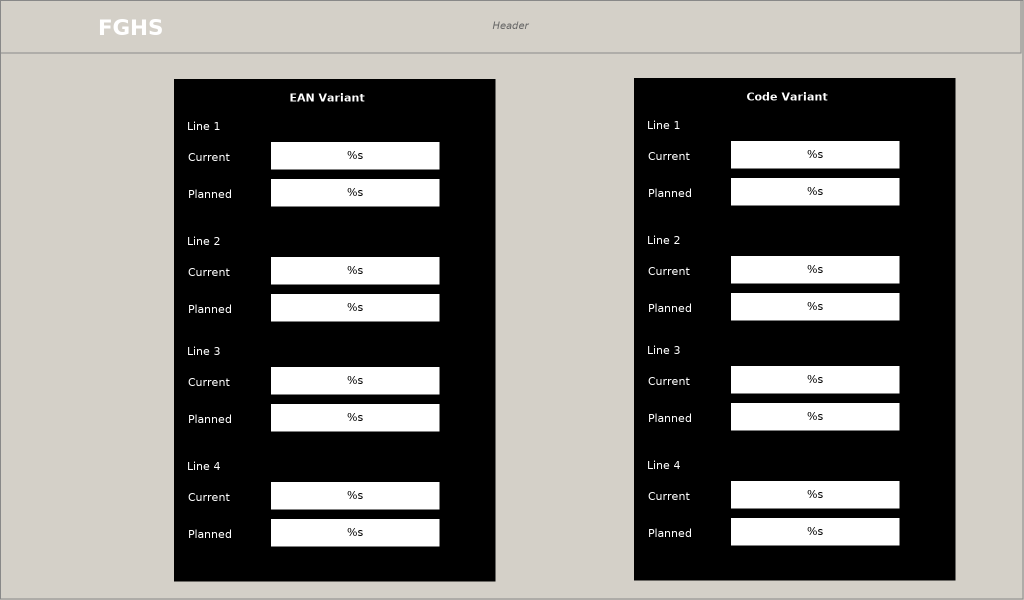
VISUALIZATION FGHS_1  // 1024x600
    Frame (0,-2 1021x55)
        shows Header()
    RoundedRectangle (174,79 321x502)
    Label (214,78 227x40), "EAN Variant"
    Label (185,140 78x35), "Current"
    RoundedRectangle (270,141 170x29), "%s", text variable: Status_GVL.arCurrent_EAN[1]
        OnMouseClick: write Status_GVL.RecipeLine[1].EANVariant via Default
    Label (185,177 78x35), "Planned"
    RoundedRectangle (270,178 170x29), "%s", text variable: Status_GVL.arPlanned_EAN[1]
    Label (95,15 250x25), "FGHS"
    Label (184,109 78x35), "Line 1"
    Label (185,255 78x35), "Current"
    RoundedRectangle (270,256 170x29), "%s", text variable: Status_GVL.arCurrent_EAN[2]
        OnMouseClick: write Status_GVL.RecipeLine[2].EANVariant via Default
    Label (185,292 78x35), "Planned"
    RoundedRectangle (270,293 170x29), "%s", text variable: Status_GVL.arPlanned_EAN[2]
    Label (184,224 78x35), "Line 2"
    Label (185,365 78x35), "Current"
    RoundedRectangle (270,366 170x29), "%s", text variable: Status_GVL.arCurrent_EAN[3]
        OnMouseClick: write Status_GVL.RecipeLine[3].EANVariant via Default
    Label (185,402 78x35), "Planned"
    RoundedRectangle (270,403 170x29), "%s", text variable: Status_GVL.arPlanned_EAN[3]
    Label (184,334 78x35), "Line 3"
    Label (185,480 78x35), "Current"
    RoundedRectangle (270,481 170x29), "%s", text variable: Status_GVL.arCurrent_EAN[4]
        OnMouseClick: write Status_GVL.RecipeLine[4].EANVariant via Default
    Label (185,517 78x35), "Planned"
    RoundedRectangle (270,518 170x29), "%s", text variable: Status_GVL.arPlanned_EAN[4]
    Label (184,449 78x35), "Line 4"
    RoundedRectangle (634,78 321x502)
    Label (674,77 227x40), "Code Variant"
    Label (645,139 78x35), "Current"
    RoundedRectangle (730,140 170x29), "%s", text variable: Status_GVL.arCurrent_CodeVariant[1]
        OnMouseClick: write Status_GVL.RecipeLine[1].CodeVariant via Default
    Label (645,176 78x35), "Planned"
    RoundedRectangle (730,177 170x29), "%s", text variable: Status_GVL.arPlanned_CodeVariant[1]
    Label (644,108 78x35), "Line 1"
    Label (645,254 78x35), "Current"
    RoundedRectangle (730,255 170x29), "%s", text variable: Status_GVL.arCurrent_CodeVariant[2]
        OnMouseClick: write Status_GVL.RecipeLine[2].CodeVariant via Default
    Label (645,291 78x35), "Planned"
    RoundedRectangle (730,292 170x29), "%s", text variable: Status_GVL.arPlanned_CodeVariant[2]
    Label (644,223 78x35), "Line 2"
    Label (645,364 78x35), "Current"
    RoundedRectangle (730,365 170x29), "%s", text variable: Status_GVL.arCurrent_CodeVariant[3]
        OnMouseClick: write Status_GVL.RecipeLine[3].CodeVariant via Default
    Label (645,401 78x35), "Planned"
    RoundedRectangle (730,402 170x29), "%s", text variable: Status_GVL.arPlanned_CodeVariant[3]
    Label (644,333 78x35), "Line 3"
    Label (645,479 78x35), "Current"
    RoundedRectangle (730,480 170x29), "%s", text variable: Status_GVL.arCurrent_CodeVariant[4]
        OnMouseClick: write Status_GVL.RecipeLine[4].CodeVariant via Default
    Label (645,516 78x35), "Planned"
    RoundedRectangle (730,517 170x29), "%s", text variable: Status_GVL.arPlanned_CodeVariant[4]
    Label (644,448 78x35), "Line 4"
END_VISUALIZATION

(* stored: Version 1.1.0.1, ProductVersion 3.1.4024.12
   Visu FGHS_1: Id {31d02872-55a1-450c-84ed-16608a4e7188} *)
